(* CODESYS project CtaAppModBusSpezifikation_1.0.0.0.library
   Description: ModbusSpezifikation Library der CTA
   Version: 1.0.0.0
   Title: CtaAppModbusSpezifikation
   Author: SIS
   Company: CTA
   DocFormat: reStructuredText
   Placeholder: CtaAppModbusSpezifikation
   CompiledLibraryCompatibilityVersion: CODESYS V3.5 SP16 Patch 3
   LanguageModelAttribute: qualified-access-only
   DefaultNamespace: CtaAppModbusSpezifikation

Project tree, tasks and I/O mapping:
  libraries: Standard, 3.5.18.0 (System); CtaAppBmk, 1.0.0.0 (CTA); VisuSymbols, 4.5.0.0 (System); VisuDialogs, * (System); CtaAppModbus, 1.0.0.0 (CTA)
  40 Visualizations/
  30 Program Organization Units/
    MODBUS SPEZIFIKATION/
      function fcModBusSpezifikation [ST]
      function fcModBusAdrBmk [ST]
  00000000-0000-0000-0000-000000000000|D:\CoDeSys\LibrariesV3\trunk\Intern\CAA\CAA Template\3.4.0.0 draft\Placeholder.xml
  00000000-0000-0000-0000-000000000000|D:\CoDeSys\LibrariesV3\trunk\Intern\CAA\CAA Template\3.2.0.3 draft\Prefix.pdf
  00000000-0000-0000-0000-000000000000|D:\CoDeSys\LibrariesV3\trunk\Intern\CAA\CAA Template\3.5.2.0 draft\Placeholder.xml
  20 Structs/
  50 Images/
  10 Documenation/
    global variables VersionHistory
    global variables readMe
  21 Interface/
    MODBUS SPEZIFIKATION/
      interface ITF_MODBUS_SPEZIFIKATION: proModbusStateWord
  11 Library Parameter/
  12 Konstanten/
  60 Textlisten/
  13 Globale Variablen/
  text list GlobalTextList
*)

// 10 Documenation/VersionHistory
(* 

.. image:: ../../Images/CTA_Logo.jpg
   :align: right
   :width: 15% 

**Vorlage**   


============ =========== =========== ============================================
**Date**     **Version** **Author**  **Change**
------------ ----------- ----------- --------------------------------------------
04.03.2021   0.0.0.0     SIS         Vorlage erstellt

============ =========== =========== ============================================


*)
VAR_GLOBAL
    stInfo : STRING:= '0.0.0.0, Vorlage, CTA';
END_VAR

// 10 Documenation/readMe
(*

**ReadMe**
 
|	**Empfehlung**
|
|	Dokumentrieren Sie die Library für eine nachhaltige Entwicklung
|     
| *Beispiel* 
|
| Dies ist die Vorlage Library der CTA. Erstellen Sie ihre Library anhand dieser Vorlage.
*)

VAR_GLOBAL
    xReadMeDone              :   BOOL;
END_VAR

// 21 Interface/MODBUS SPEZIFIKATION/ITF_MODBUS_SPEZIFIKATION
INTERFACE ITF_MODBUS_SPEZIFIKATION EXTENDS CtaAppBmk.ITF_BMK;

{warning disable C0410}
PROPERTY proModbusStateWord : REFERENCE TO ARRAY[0..3] OF WORD
{warning restore C0410}
GET
END_GET
END_PROPERTY

END_INTERFACE

// 30 Program Organization Units/MODBUS SPEZIFIKATION/fcModBusSpezifikation
FUNCTION fcModBusSpezifikation : BOOL
VAR_INPUT
	ITF_SERVER					:	CtaAppModbus.ITF_SERVER;
	ITF_MODBUS_SPEZIFIKATION	:	ITF_MODBUS_SPEZIFIKATION;
END_VAR
VAR
	wAdr		:	WORD;
END_VAR

IF __QUERYINTERFACE(ITF_SERVER,ITF_SERVER) AND __QUERYINTERFACE(ITF_MODBUS_SPEZIFIKATION,ITF_MODBUS_SPEZIFIKATION) THEN
	wAdr := fcModBusAdrBmk(ITF_MODBUS_SPEZIFIKATION);	
	IF wAdr <> 0 THEN
		ITF_SERVER.metSetInputRegister(wAdr + 0, ITF_MODBUS_SPEZIFIKATION.proModbusStateWord[0]);
		ITF_SERVER.metSetInputRegister(wAdr + 1, ITF_MODBUS_SPEZIFIKATION.proModbusStateWord[1]);
		ITF_SERVER.metSetInputRegister(wAdr + 2, ITF_MODBUS_SPEZIFIKATION.proModbusStateWord[2]);
		ITF_SERVER.metSetInputRegister(wAdr + 3, ITF_MODBUS_SPEZIFIKATION.proModbusStateWord[3]);
	END_IF
END_IF;

END_FUNCTION

// 30 Program Organization Units/MODBUS SPEZIFIKATION/fcModBusAdrBmk
FUNCTION fcModBusAdrBmk : WORD
VAR_INPUT
	ITF_BMK	:	CtaAppBmk.ITF_BMK;
END_VAR
VAR
	stBMK	:	STRING(7);
	iLen	:	INT;
	wFu		:	WORD;
	wBl		:	WORD;
	wDe		:	WORD;
END_VAR

(* Not Valid *)
fcModBusAdrBmk := 0;
IF __QUERYINTERFACE(ITF_BMK,ITF_BMK) THEN
	IF ITF_BMK.proGetObjectId <> '' THEN
		stBMK := ITF_BMK.proGetBMK;
		(* Check if Valid BMK min 5 Charakters *)
		IF Standard.LEN(stBMK) = 7 THEN
			iLen := TO_INT(Standard.LEN(stBMK));	
			wFu := TO_WORD(Standard.LEFT(stBMK,TO_INT(-4 + iLen)));
			wBl := TO_WORD(Standard.MID(stBMK,2,(-2 + iLen)));
			wDe := TO_WORD(Standard.RIGHT(stBMK,1));
			(* Check if first Charakters are >= 100 & <= 899*)
			IF wFu >= 100 AND wFu <= 899 THEN
				IF wBl >= 1 AND wBl <= 99 THEN
					IF wDe >= 1 AND wDe <= 2 THEN
						(* Adr 100000 - 297802*)
						fcModBusAdrBmk := 1000 + ((wFu-100)*80) + ((wBl-1)*8) + ((wDe-1)*4);
					END_IF;
				END_IF;
			END_IF;
		END_IF;
	END_IF;
END_IF

END_FUNCTION
